TYPE ST_StatusDevices :
STRUCT

	sLivingRoom						: ST_LivingRoomDevices;
	sBedroom						: ST_BedroomDevices;

END_STRUCT
END_TYPE

(* stored: Version 1.1.0.1, ProductVersion 3.1.4024.12
   DUT ST_StatusDevices: Id {8d3dcedd-6fab-477c-af80-c8bb012f79d8} *)
